PROGRAM P2_00_MAIN
VAR
	tonFlapReset			:TON;
END_VAR

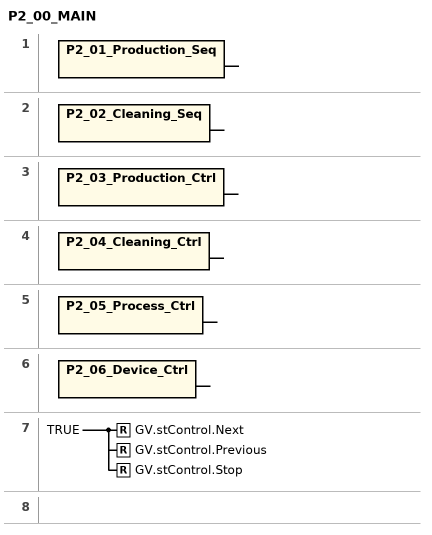
// NETWORK 1
P2_01_Production_Seq();

// NETWORK 2
P2_02_Cleaning_Seq();

// NETWORK 3
P2_03_Production_Ctrl();

// NETWORK 4
P2_04_Cleaning_Ctrl();

// NETWORK 5
P2_05_Process_Ctrl();

// NETWORK 6
P2_06_Device_Ctrl();

// NETWORK 7
GV.stControl.Next R= TRUE;
GV.stControl.Previous R= TRUE;
GV.stControl.Stop R= TRUE;

// NETWORK 8

END_PROGRAM

(* stored: Version 1.1.0.1
   POU P2_00_MAIN: Id {ca4a7650-0b0a-4fcf-be5c-8c1e0434016e}, SpecialFunc None *)
